% RSLogix 500 project alarm_and_notifcations.RSS, saved by version 9.00.00.04 %
PROJECT "UNTITLED"    % processor: Bul.1763 MicroLogix 1100 Series A %

PROGRAM FILES
  LAD 2 "MAIN"  10 rungs
  LAD 3 "D INPUT"  9 rungs
  LAD 4 "D OUTPUT"  6 rungs
  LAD 5 "A INPUT"  3 rungs
  LAD 6 "A OUTPUT"  2 rungs
  LAD 7 "CONTROLS"  13 rungs
  LAD 8 "ALARMS"  21 rungs
  LAD 9 "DISPLAY"  2 rungs

DATA FILES
  O0 OUTPUT  6 elements
  I1 INPUT  18 elements
  S2 STATUS  66 elements
  B3 BINARY  8 elements
  T4 TIMER  8 elements
  C5 COUNTER  1 elements
  R6 CONTROL  1 elements
  N7 INTEGER  12 elements
  F8 FLOAT  3 elements
  PD9 TEMP  1 elements

LADDER 2 "MAIN"
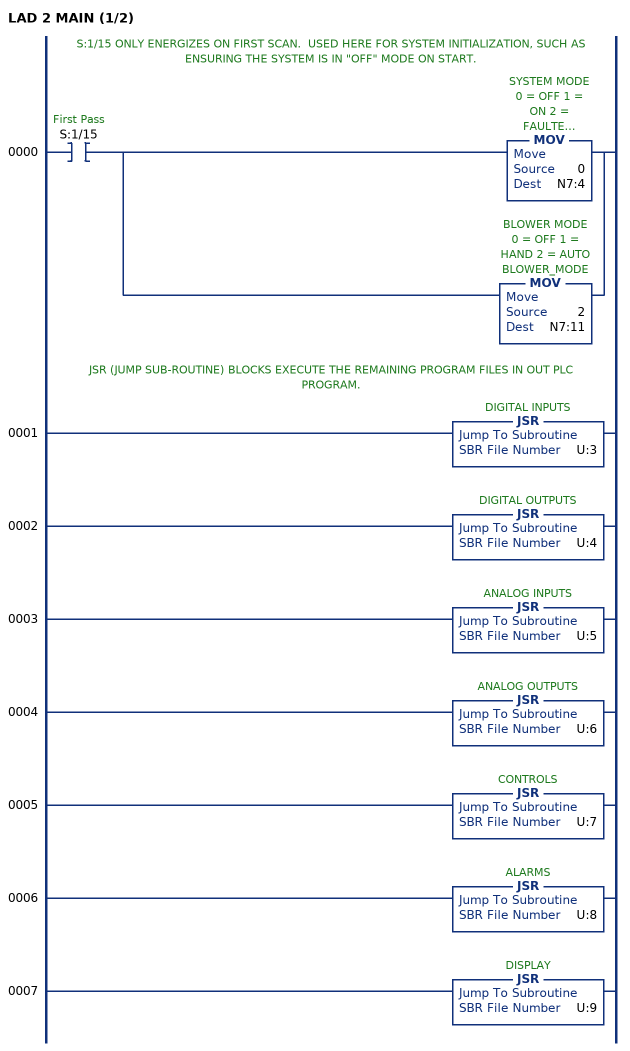
% Rung: 0 %
% S:1/15 ONLY ENERGIZES ON FIRST SCAN.  USED HERE FOR SYSTEM INITIALIZATION, SUCH AS ENSURING THE SYSTEM IS IN "OFF" MODE ON START. %
SOR XIC S:1/15 BST MOV 0 N7:4 NXB MOV 2 N7:11 BND EOR
%   S:1/15  "First Pass" %
%   N7:4  SYSTEM_MODE  "SYSTEM MODE 0 = OFF 1 = ON 2 = FAULTED" %
%   N7:11  BLOWER_MODE  "BLOWER MODE 0 = OFF 1 = HAND 2 = AUTO" %
% Rung: 1 %
% JSR (JUMP SUB-ROUTINE) BLOCKS EXECUTE THE REMAINING PROGRAM FILES IN OUT PLC PROGRAM. %
SOR JSR U:3 EOR
%   U:3  "DIGITAL INPUTS" %
% Rung: 2 %
SOR JSR U:4 EOR
%   U:4  "DIGITAL OUTPUTS" %
% Rung: 3 %
SOR JSR U:5 EOR
%   U:5  "ANALOG INPUTS" %
% Rung: 4 %
SOR JSR U:6 EOR
%   U:6  "ANALOG OUTPUTS" %
% Rung: 5 %
SOR JSR U:7 EOR
%   U:7  "CONTROLS" %
% Rung: 6 %
SOR JSR U:8 EOR
%   U:8  "ALARMS" %
% Rung: 7 %
SOR JSR U:9 EOR
%   U:9  "DISPLAY" %

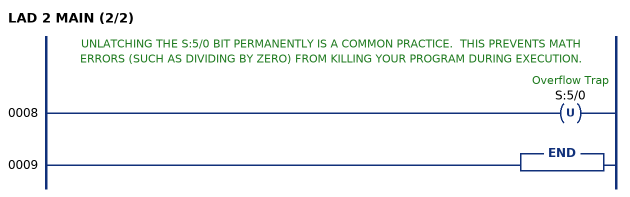
% Rung: 8 %
% UNLATCHING THE S:5/0 BIT PERMANENTLY IS A COMMON PRACTICE.  THIS PREVENTS MATH ERRORS (SUCH AS DIVIDING BY ZERO) FROM KILLING YOUR PROGRAM DURING EXECUTION. %
SOR OTU S:5/0 EOR
%   S:5/0  "Overflow Trap" %
% Rung: 9 %
SOR END EOR

LADDER 3 "D INPUT"
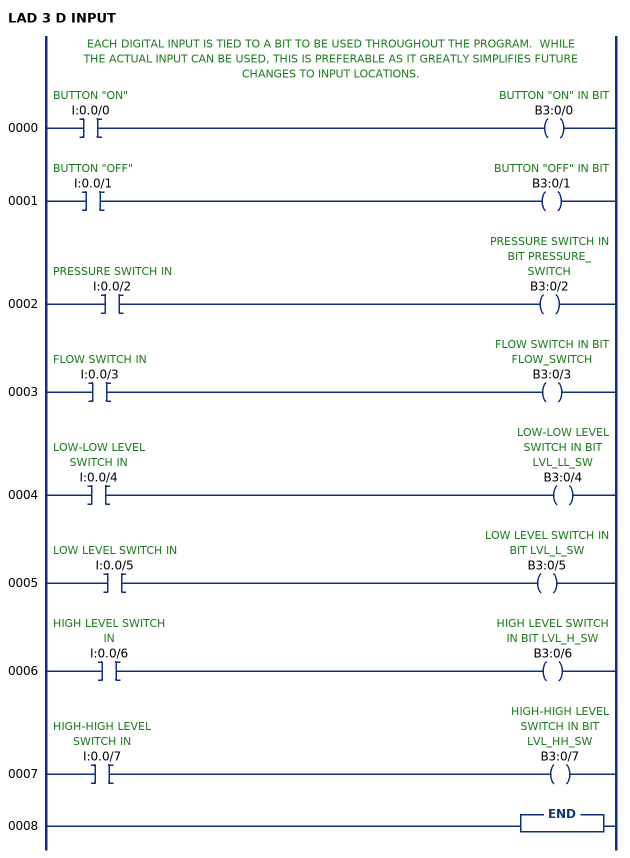
% Rung: 0 %
% EACH DIGITAL INPUT IS TIED TO A BIT TO BE USED THROUGHOUT THE PROGRAM.  WHILE THE ACTUAL INPUT CAN BE USED, THIS IS PREFERABLE AS IT GREATLY SIMPLIFIES FUTURE CHANGES TO INPUT LOCATIONS. %
SOR XIC I:0.0/0 OTE B3:0/0 EOR
%   I:0.0/0  "BUTTON "ON"" %
%   B3:0/0  "BUTTON "ON" IN BIT" %
% Rung: 1 %
SOR XIC I:0.0/1 OTE B3:0/1 EOR
%   I:0.0/1  "BUTTON "OFF"" %
%   B3:0/1  "BUTTON "OFF" IN BIT" %
% Rung: 2 %
SOR XIC I:0.0/2 OTE B3:0/2 EOR
%   I:0.0/2  "PRESSURE SWITCH IN" %
%   B3:0/2  PRESSURE_SWITCH  "PRESSURE SWITCH IN BIT" %
% Rung: 3 %
SOR XIC I:0.0/3 OTE B3:0/3 EOR
%   I:0.0/3  "FLOW SWITCH IN" %
%   B3:0/3  FLOW_SWITCH  "FLOW SWITCH IN BIT" %
% Rung: 4 %
SOR XIC I:0.0/4 OTE B3:0/4 EOR
%   I:0.0/4  "LOW-LOW LEVEL SWITCH IN" %
%   B3:0/4  LVL_LL_SW  "LOW-LOW LEVEL SWITCH IN BIT" %
% Rung: 5 %
SOR XIC I:0.0/5 OTE B3:0/5 EOR
%   I:0.0/5  "LOW LEVEL SWITCH IN" %
%   B3:0/5  LVL_L_SW  "LOW LEVEL SWITCH IN BIT" %
% Rung: 6 %
SOR XIC I:0.0/6 OTE B3:0/6 EOR
%   I:0.0/6  "HIGH LEVEL SWITCH IN" %
%   B3:0/6  LVL_H_SW  "HIGH LEVEL SWITCH IN BIT" %
% Rung: 7 %
SOR XIC I:0.0/7 OTE B3:0/7 EOR
%   I:0.0/7  "HIGH-HIGH LEVEL SWITCH IN" %
%   B3:0/7  LVL_HH_SW  "HIGH-HIGH LEVEL SWITCH IN BIT" %
% Rung: 8 %
SOR END EOR

LADDER 4 "D OUTPUT"
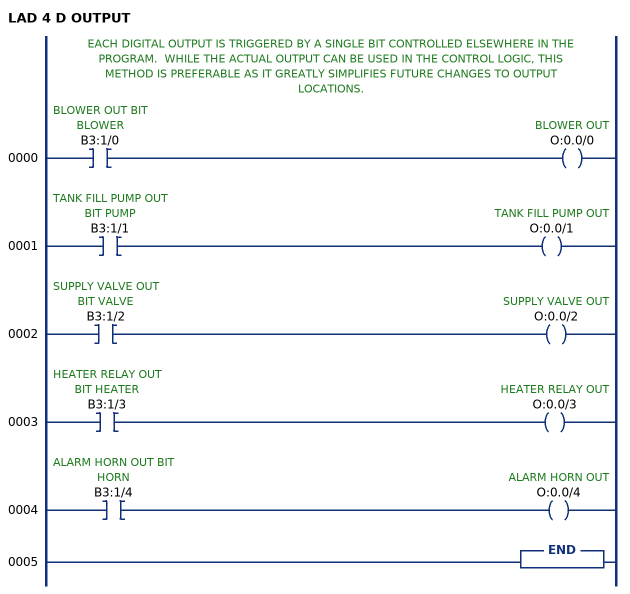
% Rung: 0 %
% EACH DIGITAL OUTPUT IS TRIGGERED BY A SINGLE BIT CONTROLLED ELSEWHERE IN THE PROGRAM.  WHILE THE ACTUAL OUTPUT CAN BE USED IN THE CONTROL LOGIC, THIS METHOD IS PREFERABLE AS IT GREATLY SIMPLIFIES FUTURE CHANGES TO OUTPUT LOCATIONS. %
SOR XIC B3:1/0 OTE O:0.0/0 EOR
%   B3:1/0  BLOWER  "BLOWER OUT BIT" %
%   O:0.0/0  "BLOWER OUT" %
% Rung: 1 %
SOR XIC B3:1/1 OTE O:0.0/1 EOR
%   B3:1/1  PUMP  "TANK FILL PUMP OUT BIT" %
%   O:0.0/1  "TANK FILL PUMP OUT" %
% Rung: 2 %
SOR XIC B3:1/2 OTE O:0.0/2 EOR
%   B3:1/2  VALVE  "SUPPLY VALVE OUT BIT" %
%   O:0.0/2  "SUPPLY VALVE OUT" %
% Rung: 3 %
SOR XIC B3:1/3 OTE O:0.0/3 EOR
%   B3:1/3  HEATER  "HEATER RELAY OUT BIT" %
%   O:0.0/3  "HEATER RELAY OUT" %
% Rung: 4 %
SOR XIC B3:1/4 OTE O:0.0/4 EOR
%   B3:1/4  HORN  "ALARM HORN OUT BIT" %
%   O:0.0/4  "ALARM HORN OUT" %
% Rung: 5 %
SOR END EOR

LADDER 5 "A INPUT"
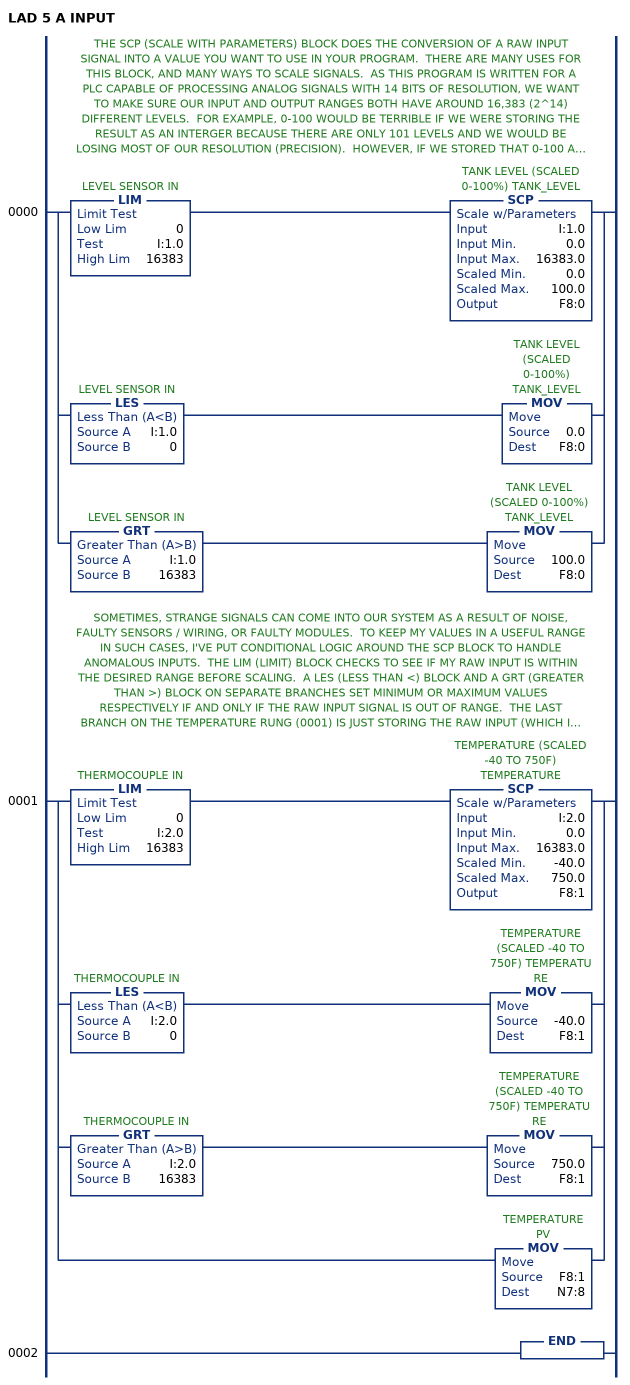
% Rung: 0 %
% THE SCP (SCALE WITH PARAMETERS) BLOCK DOES THE CONVERSION OF A RAW INPUT SIGNAL INTO A VALUE YOU WANT TO USE IN YOUR PROGRAM.  THERE ARE MANY USES FOR THIS BLOCK, AND MANY WAYS TO SCALE SIGNALS.  AS THIS PROGRAM IS WRITTEN FOR A PLC CAPABLE OF PROCESSING ANALOG SIGNALS WITH 14 BITS OF RESOLUTION, WE WANT TO MAKE SURE OUR INPUT AND OUTPUT RANGES BOTH HAVE AROUND 16,383 (2^14) DIFFERENT LEVELS.  FOR EXAMPLE, 0-100 WOULD BE TERRIBLE IF WE WERE STORING THE RESULT AS AN INTERGER BECAUSE THERE ARE ONLY 101 LEVELS AND WE WOULD BE LOSING MOST OF OUR RESOLUTION (PRECISION).  HOWEVER, IF WE STORED THAT 0-100 AS A FLOAT WITH TWO DECIMAL PLACES, IT'S BETTER BECAUSE WE THEN HAVE 10,001 LEVELS.  HOWEVER, THIS STILL ISN'T IDEAL. %
SOR BST LIM 0 I:1.0 16383 SCP I:1.0 0.0 16383.0 0.0 100.0 F8:0 NXB LES I:1.0 0 MOV 0.0 F8:0 NXB GRT I:1.0 16383 MOV 100.0 F8:0 BND EOR
%   I:1.0  "LEVEL SENSOR IN" %
%   F8:0  TANK_LEVEL  "TANK LEVEL (SCALED 0-100%)" %
% Rung: 1 %
% SOMETIMES, STRANGE SIGNALS CAN COME INTO OUR SYSTEM AS A RESULT OF NOISE, FAULTY SENSORS / WIRING, OR FAULTY MODULES.  TO KEEP MY VALUES IN A USEFUL RANGE IN SUCH CASES, I'VE PUT CONDITIONAL LOGIC AROUND THE SCP BLOCK TO HANDLE ANOMALOUS INPUTS.  THE LIM (LIMIT) BLOCK CHECKS TO SEE IF MY RAW INPUT IS WITHIN THE DESIRED RANGE BEFORE SCALING.  A LES (LESS THAN <) BLOCK AND A GRT (GREATER THAN >) BLOCK ON SEPARATE BRANCHES SET MINIMUM OR MAXIMUM VALUES RESPECTIVELY IF AND ONLY IF THE RAW INPUT SIGNAL IS OUT OF RANGE.  THE LAST BRANCH ON THE TEMPERATURE RUNG (0001) IS JUST STORING THE RAW INPUT (WHICH IS ALREADY SCALED FOR PID 0-16383) TO AN INTERGER REGISTER IN MEMORY FOR USE IN A PID CONTROL LOOP.  THIS PREVENTS ME FROM REFERRING TO THE ACTUAL INPUT WITHIN THE REST OF THE PROGRAM.  THUS, IF IN THE FUTURE WE NEED TO REMAP OUR IO, WE ONLY HAVE TO MAKE CHANGES IN THE IO PROGRAM FILES INSTEAD OF HUNTING EACH ADDRESS THROUGHOUT THE ENTIRE PROGRAM. %
SOR BST LIM 0 I:2.0 16383 SCP I:2.0 0.0 16383.0 -40.0 750.0 F8:1 NXB LES I:2.0 0 MOV -40.0 F8:1 NXB GRT I:2.0 16383 MOV 750.0 F8:1 NXB MOV F8:1 N7:8 BND EOR
%   I:2.0  "THERMOCOUPLE IN" %
%   F8:1  TEMPERATURE  "TEMPERATURE (SCALED -40 TO 750F)" %
%   N7:8  "TEMPERATURE PV" %
% Rung: 2 %
SOR END EOR

LADDER 6 "A OUTPUT"
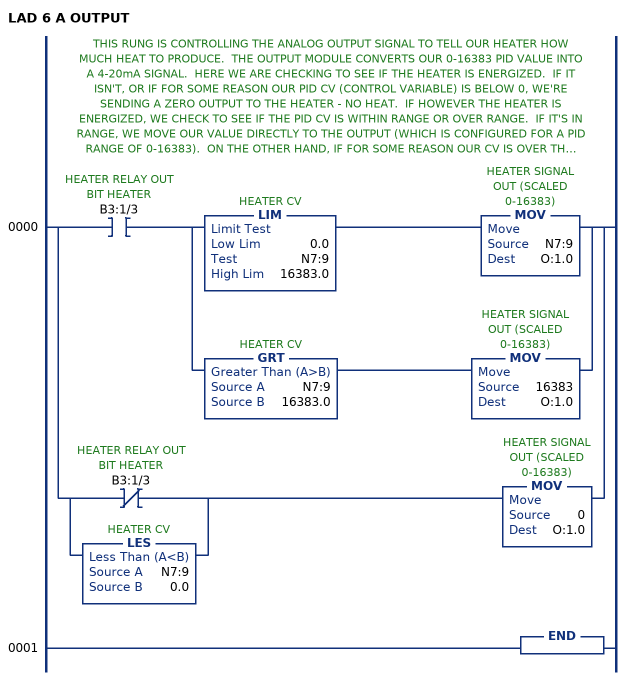
% Rung: 0 %
% THIS RUNG IS CONTROLLING THE ANALOG OUTPUT SIGNAL TO TELL OUR HEATER HOW MUCH HEAT TO PRODUCE.  THE OUTPUT MODULE CONVERTS OUR 0-16383 PID VALUE INTO A 4-20mA SIGNAL.  HERE WE ARE CHECKING TO SEE IF THE HEATER IS ENERGIZED.  IF IT ISN'T, OR IF FOR SOME REASON OUR PID CV (CONTROL VARIABLE) IS BELOW 0, WE'RE SENDING A ZERO OUTPUT TO THE HEATER - NO HEAT.  IF HOWEVER THE HEATER IS ENERGIZED, WE CHECK TO SEE IF THE PID CV IS WITHIN RANGE OR OVER RANGE.  IF IT'S IN RANGE, WE MOVE OUR VALUE DIRECTLY TO THE OUTPUT (WHICH IS CONFIGURED FOR A PID RANGE OF 0-16383).  ON THE OTHER HAND, IF FOR SOME REASON OUR CV IS OVER THE RANGE, WE'RE MOVING A MAXIMUM ACCEPTABLE VALUE TO THE OUTPUT. %
SOR BST XIC B3:1/3 BST LIM 0.0 N7:9 16383.0 MOV N7:9 O:1.0 NXB GRT N7:9 16383.0 MOV 16383 O:1.0 BND NXB BST XIO B3:1/3 NXB LES N7:9 0.0 BND MOV 0 O:1.0 BND EOR
%   B3:1/3  HEATER  "HEATER RELAY OUT BIT" %
%   N7:9  "HEATER CV" %
%   O:1.0  "HEATER SIGNAL OUT (SCALED 0-16383)" %
% Rung: 1 %
SOR END EOR

LADDER 7 "CONTROLS"
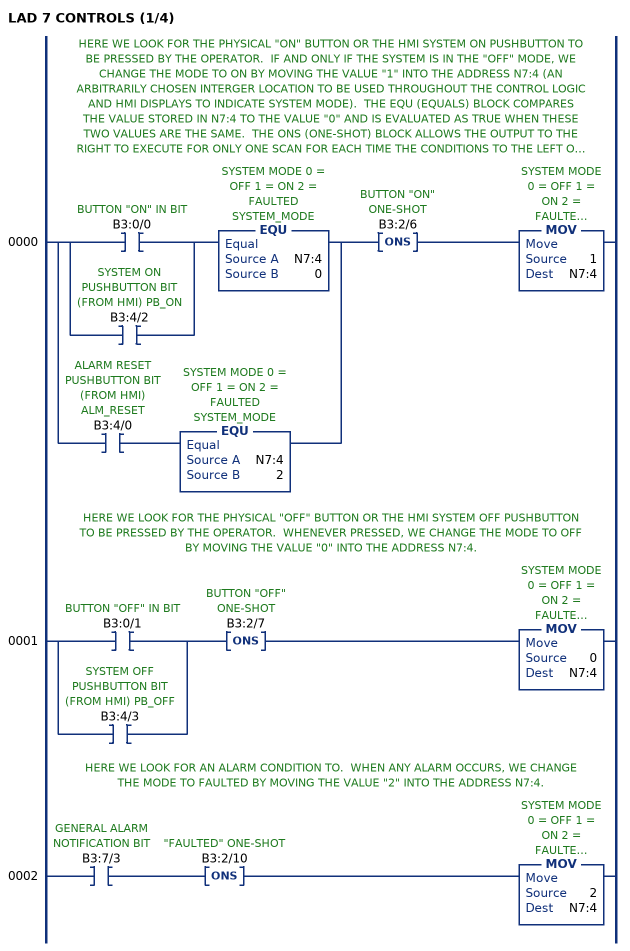
% Rung: 0 %
% HERE WE LOOK FOR THE PHYSICAL "ON" BUTTON OR THE HMI SYSTEM ON PUSHBUTTON TO BE PRESSED BY THE OPERATOR.  IF AND ONLY IF THE SYSTEM IS IN THE "OFF" MODE, WE CHANGE THE MODE TO ON BY MOVING THE VALUE "1" INTO THE ADDRESS N7:4 (AN ARBITRARILY CHOSEN INTERGER LOCATION TO BE USED THROUGHOUT THE CONTROL LOGIC AND HMI DISPLAYS TO INDICATE SYSTEM MODE).  THE EQU (EQUALS) BLOCK COMPARES THE VALUE STORED IN N7:4 TO THE VALUE "0" AND IS EVALUATED AS TRUE WHEN THESE TWO VALUES ARE THE SAME.  THE ONS (ONE-SHOT) BLOCK ALLOWS THE OUTPUT TO THE RIGHT TO EXECUTE FOR ONLY ONE SCAN FOR EACH TIME THE CONDITIONS TO THE LEFT OF THE BLOCK ARE ALL TRUE. %
SOR BST BST XIC B3:0/0 NXB XIC B3:4/2 BND EQU N7:4 0 NXB XIC B3:4/0 EQU N7:4 2 BND ONS B3:2/6 MOV 1 N7:4 EOR
%   B3:0/0  "BUTTON "ON" IN BIT" %
%   B3:4/2  PB_ON  "SYSTEM ON PUSHBUTTON BIT (FROM HMI)" %
%   N7:4  SYSTEM_MODE  "SYSTEM MODE 0 = OFF 1 = ON 2 = FAULTED" %
%   B3:4/0  ALM_RESET  "ALARM RESET PUSHBUTTON BIT (FROM HMI)" %
%   B3:2/6  "BUTTON "ON" ONE-SHOT" %
% Rung: 1 %
% HERE WE LOOK FOR THE PHYSICAL "OFF" BUTTON OR THE HMI SYSTEM OFF PUSHBUTTON TO BE PRESSED BY THE OPERATOR.  WHENEVER PRESSED, WE CHANGE THE MODE TO OFF BY MOVING THE VALUE "0" INTO THE ADDRESS N7:4. %
SOR BST XIC B3:0/1 NXB XIC B3:4/3 BND ONS B3:2/7 MOV 0 N7:4 EOR
%   B3:0/1  "BUTTON "OFF" IN BIT" %
%   B3:4/3  PB_OFF  "SYSTEM OFF PUSHBUTTON BIT (FROM HMI)" %
%   B3:2/7  "BUTTON "OFF" ONE-SHOT" %
%   N7:4  SYSTEM_MODE  "SYSTEM MODE 0 = OFF 1 = ON 2 = FAULTED" %
% Rung: 2 %
% HERE WE LOOK FOR AN ALARM CONDITION TO.  WHEN ANY ALARM OCCURS, WE CHANGE THE MODE TO FAULTED BY MOVING THE VALUE "2" INTO THE ADDRESS N7:4. %
SOR XIC B3:7/3 ONS B3:2/10 MOV 2 N7:4 EOR
%   B3:7/3  "GENERAL ALARM NOTIFICATION BIT" %
%   B3:2/10  ""FAULTED" ONE-SHOT" %
%   N7:4  SYSTEM_MODE  "SYSTEM MODE 0 = OFF 1 = ON 2 = FAULTED" %

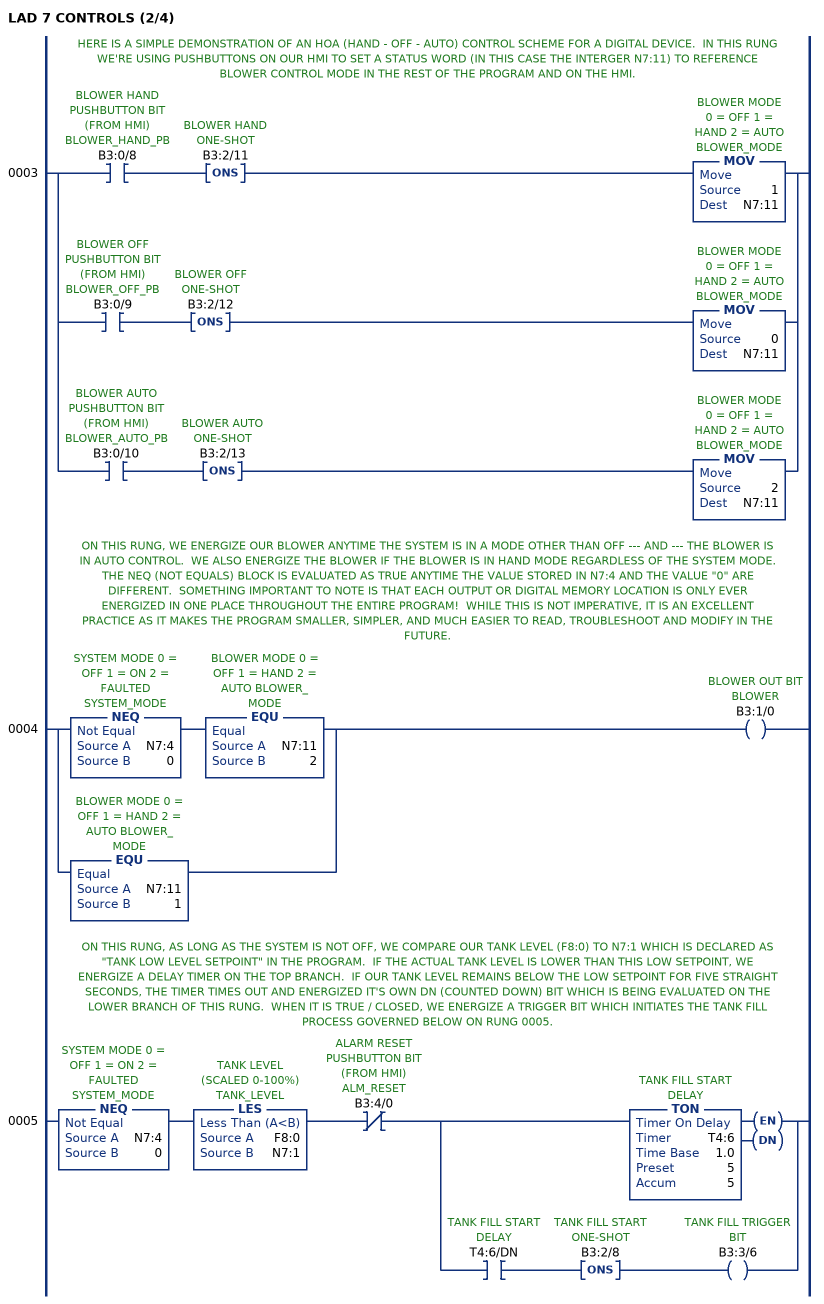
% Rung: 3 %
% HERE IS A SIMPLE DEMONSTRATION OF AN HOA (HAND - OFF - AUTO) CONTROL SCHEME FOR A DIGITAL DEVICE.  IN THIS RUNG WE'RE USING PUSHBUTTONS ON OUR HMI TO SET A STATUS WORD (IN THIS CASE THE INTERGER N7:11) TO REFERENCE BLOWER CONTROL MODE IN THE REST OF THE PROGRAM AND ON THE HMI. %
SOR BST XIC B3:0/8 ONS B3:2/11 MOV 1 N7:11 NXB XIC B3:0/9 ONS B3:2/12 MOV 0 N7:11 NXB XIC B3:0/10 ONS B3:2/13 MOV 2 N7:11 BND EOR
%   B3:0/8  BLOWER_HAND_PB  "BLOWER HAND PUSHBUTTON BIT (FROM HMI)" %
%   B3:2/11  "BLOWER HAND ONE-SHOT" %
%   N7:11  BLOWER_MODE  "BLOWER MODE 0 = OFF 1 = HAND 2 = AUTO" %
%   B3:0/9  BLOWER_OFF_PB  "BLOWER OFF PUSHBUTTON BIT (FROM HMI)" %
%   B3:2/12  "BLOWER OFF ONE-SHOT" %
%   B3:0/10  BLOWER_AUTO_PB  "BLOWER AUTO PUSHBUTTON BIT (FROM HMI)" %
%   B3:2/13  "BLOWER AUTO ONE-SHOT" %
% Rung: 4 %
% ON THIS RUNG, WE ENERGIZE OUR BLOWER ANYTIME THE SYSTEM IS IN A MODE OTHER THAN OFF --- AND --- THE BLOWER IS IN AUTO CONTROL.  WE ALSO ENERGIZE THE BLOWER IF THE BLOWER IS IN HAND MODE REGARDLESS OF THE SYSTEM MODE.  THE NEQ (NOT EQUALS) BLOCK IS EVALUATED AS TRUE ANYTIME THE VALUE STORED IN N7:4 AND THE VALUE "0" ARE DIFFERENT.  SOMETHING IMPORTANT TO NOTE IS THAT EACH OUTPUT OR DIGITAL MEMORY LOCATION IS ONLY EVER ENERGIZED IN ONE PLACE THROUGHOUT THE ENTIRE PROGRAM!  WHILE THIS IS NOT IMPERATIVE, IT IS AN EXCELLENT PRACTICE AS IT MAKES THE PROGRAM SMALLER, SIMPLER, AND MUCH EASIER TO READ, TROUBLESHOOT AND MODIFY IN THE FUTURE. %
SOR BST NEQ N7:4 0 EQU N7:11 2 NXB EQU N7:11 1 BND OTE B3:1/0 EOR
%   N7:4  SYSTEM_MODE  "SYSTEM MODE 0 = OFF 1 = ON 2 = FAULTED" %
%   N7:11  BLOWER_MODE  "BLOWER MODE 0 = OFF 1 = HAND 2 = AUTO" %
%   B3:1/0  BLOWER  "BLOWER OUT BIT" %
% Rung: 5 %
% ON THIS RUNG, AS LONG AS THE SYSTEM IS NOT OFF, WE COMPARE OUR TANK LEVEL (F8:0) TO N7:1 WHICH IS DECLARED AS "TANK LOW LEVEL SETPOINT" IN THE PROGRAM.  IF THE ACTUAL TANK LEVEL IS LOWER THAN THIS LOW SETPOINT, WE ENERGIZE A DELAY TIMER ON THE TOP BRANCH.  IF OUR TANK LEVEL REMAINS BELOW THE LOW SETPOINT FOR FIVE STRAIGHT SECONDS, THE TIMER TIMES OUT AND ENERGIZED IT'S OWN DN (COUNTED DOWN) BIT WHICH IS BEING EVALUATED ON THE LOWER BRANCH OF THIS RUNG.  WHEN IT IS TRUE / CLOSED, WE ENERGIZE A TRIGGER BIT WHICH INITIATES THE TANK FILL PROCESS GOVERNED BELOW ON RUNG 0005. %
SOR NEQ N7:4 0 LES F8:0 N7:1 XIO B3:4/0 BST TON T4:6 1.0 5 5 NXB XIC T4:6/DN ONS B3:2/8 OTE B3:3/6 BND EOR
%   N7:4  SYSTEM_MODE  "SYSTEM MODE 0 = OFF 1 = ON 2 = FAULTED" %
%   F8:0  TANK_LEVEL  "TANK LEVEL (SCALED 0-100%)" %
%   N7:1  TANK_SP_L  "TANK LOW LEVEL SETPOINT" %
%   B3:4/0  ALM_RESET  "ALARM RESET PUSHBUTTON BIT (FROM HMI)" %
%   T4:6  "TANK FILL START DELAY" %
%   B3:2/8  "TANK FILL START ONE-SHOT" %
%   B3:3/6  "TANK FILL TRIGGER BIT" %

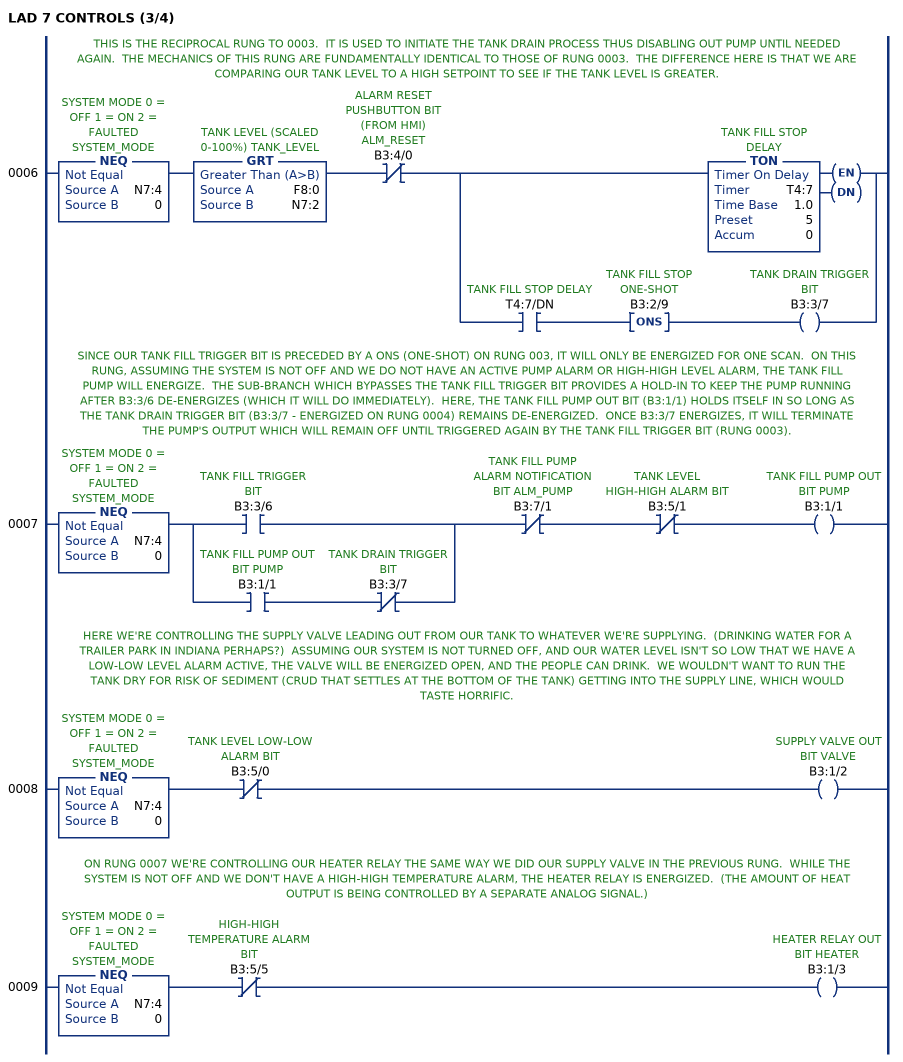
% Rung: 6 %
% THIS IS THE RECIPROCAL RUNG TO 0003.  IT IS USED TO INITIATE THE TANK DRAIN PROCESS THUS DISABLING OUT PUMP UNTIL NEEDED AGAIN.  THE MECHANICS OF THIS RUNG ARE FUNDAMENTALLY IDENTICAL TO THOSE OF RUNG 0003.  THE DIFFERENCE HERE IS THAT WE ARE COMPARING OUR TANK LEVEL TO A HIGH SETPOINT TO SEE IF THE TANK LEVEL IS GREATER. %
SOR NEQ N7:4 0 GRT F8:0 N7:2 XIO B3:4/0 BST TON T4:7 1.0 5 0 NXB XIC T4:7/DN ONS B3:2/9 OTE B3:3/7 BND EOR
%   N7:4  SYSTEM_MODE  "SYSTEM MODE 0 = OFF 1 = ON 2 = FAULTED" %
%   F8:0  TANK_LEVEL  "TANK LEVEL (SCALED 0-100%)" %
%   N7:2  TANK_SP_H  "TANK HIGH LEVEL SETPOINT" %
%   B3:4/0  ALM_RESET  "ALARM RESET PUSHBUTTON BIT (FROM HMI)" %
%   T4:7  "TANK FILL STOP DELAY" %
%   B3:2/9  "TANK FILL STOP ONE-SHOT" %
%   B3:3/7  "TANK DRAIN TRIGGER BIT" %
% Rung: 7 %
% SINCE OUR TANK FILL TRIGGER BIT IS PRECEDED BY A ONS (ONE-SHOT) ON RUNG 003, IT WILL ONLY BE ENERGIZED FOR ONE SCAN.  ON THIS RUNG, ASSUMING THE SYSTEM IS NOT OFF AND WE DO NOT HAVE AN ACTIVE PUMP ALARM OR HIGH-HIGH LEVEL ALARM, THE TANK FILL PUMP WILL ENERGIZE.  THE SUB-BRANCH WHICH BYPASSES THE TANK FILL TRIGGER BIT PROVIDES A HOLD-IN TO KEEP THE PUMP RUNNING AFTER B3:3/6 DE-ENERGIZES (WHICH IT WILL DO IMMEDIATELY).  HERE, THE TANK FILL PUMP OUT BIT (B3:1/1) HOLDS ITSELF IN SO LONG AS THE TANK DRAIN TRIGGER BIT (B3:3/7 - ENERGIZED ON RUNG 0004) REMAINS DE-ENERGIZED.  ONCE B3:3/7 ENERGIZES, IT WILL TERMINATE THE PUMP'S OUTPUT WHICH WILL REMAIN OFF UNTIL TRIGGERED AGAIN BY THE TANK FILL TRIGGER BIT (RUNG 0003). %
SOR NEQ N7:4 0 BST XIC B3:3/6 NXB XIC B3:1/1 XIO B3:3/7 BND XIO B3:7/1 XIO B3:5/1 OTE B3:1/1 EOR
%   N7:4  SYSTEM_MODE  "SYSTEM MODE 0 = OFF 1 = ON 2 = FAULTED" %
%   B3:3/6  "TANK FILL TRIGGER BIT" %
%   B3:1/1  PUMP  "TANK FILL PUMP OUT BIT" %
%   B3:3/7  "TANK DRAIN TRIGGER BIT" %
%   B3:7/1  ALM_PUMP  "TANK FILL PUMP ALARM NOTIFICATION BIT" %
%   B3:5/1  "TANK LEVEL HIGH-HIGH ALARM BIT" %
% Rung: 8 %
% HERE WE'RE CONTROLLING THE SUPPLY VALVE LEADING OUT FROM OUR TANK TO WHATEVER WE'RE SUPPLYING.  (DRINKING WATER FOR A TRAILER PARK IN INDIANA PERHAPS?)  ASSUMING OUR SYSTEM IS NOT TURNED OFF, AND OUR WATER LEVEL ISN'T SO LOW THAT WE HAVE A LOW-LOW LEVEL ALARM ACTIVE, THE VALVE WILL BE ENERGIZED OPEN, AND THE PEOPLE CAN DRINK.  WE WOULDN'T WANT TO RUN THE TANK DRY FOR RISK OF SEDIMENT (CRUD THAT SETTLES AT THE BOTTOM OF THE TANK) GETTING INTO THE SUPPLY LINE, WHICH WOULD TASTE HORRIFIC. %
SOR NEQ N7:4 0 XIO B3:5/0 OTE B3:1/2 EOR
%   N7:4  SYSTEM_MODE  "SYSTEM MODE 0 = OFF 1 = ON 2 = FAULTED" %
%   B3:5/0  "TANK LEVEL LOW-LOW ALARM BIT" %
%   B3:1/2  VALVE  "SUPPLY VALVE OUT BIT" %
% Rung: 9 %
% ON RUNG 0007 WE'RE CONTROLLING OUR HEATER RELAY THE SAME WAY WE DID OUR SUPPLY VALVE IN THE PREVIOUS RUNG.  WHILE THE SYSTEM IS NOT OFF AND WE DON'T HAVE A HIGH-HIGH TEMPERATURE ALARM, THE HEATER RELAY IS ENERGIZED.  (THE AMOUNT OF HEAT OUTPUT IS BEING CONTROLLED BY A SEPARATE ANALOG SIGNAL.) %
SOR NEQ N7:4 0 XIO B3:5/5 OTE B3:1/3 EOR
%   N7:4  SYSTEM_MODE  "SYSTEM MODE 0 = OFF 1 = ON 2 = FAULTED" %
%   B3:5/5  "HIGH-HIGH TEMPERATURE ALARM BIT" %
%   B3:1/3  HEATER  "HEATER RELAY OUT BIT" %

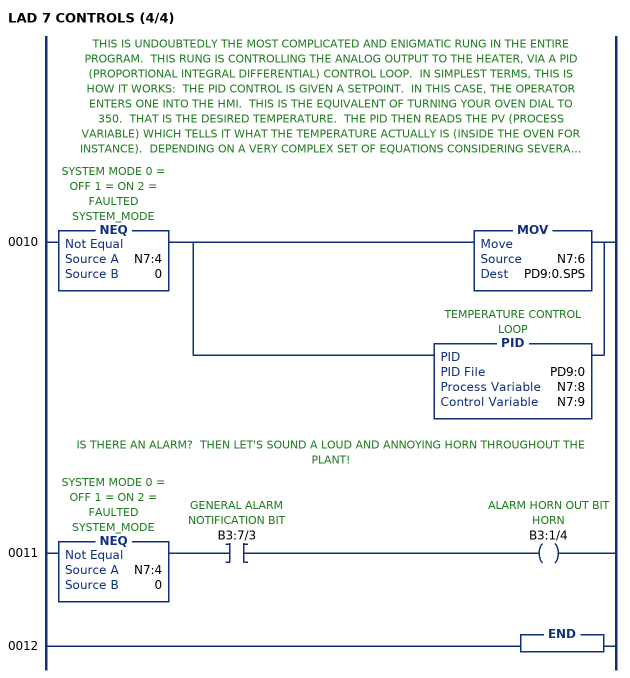
% Rung: 10 %
% THIS IS UNDOUBTEDLY THE MOST COMPLICATED AND ENIGMATIC RUNG IN THE ENTIRE PROGRAM.  THIS RUNG IS CONTROLLING THE ANALOG OUTPUT TO THE HEATER, VIA A PID (PROPORTIONAL INTEGRAL DIFFERENTIAL) CONTROL LOOP.  IN SIMPLEST TERMS, THIS IS HOW IT WORKS:  THE PID CONTROL IS GIVEN A SETPOINT.  IN THIS CASE, THE OPERATOR ENTERS ONE INTO THE HMI.  THIS IS THE EQUIVALENT OF TURNING YOUR OVEN DIAL TO 350.  THAT IS THE DESIRED TEMPERATURE.  THE PID THEN READS THE PV (PROCESS VARIABLE) WHICH TELLS IT WHAT THE TEMPERATURE ACTUALLY IS (INSIDE THE OVEN FOR INSTANCE).  DEPENDING ON A VERY COMPLEX SET OF EQUATIONS CONSIDERING SEVERAL PROGRAMMER-CONFIGURABLE VARIABLES TOO COMPLEX TO GET INTO IN THIS TUTORIAL, IT ADJUSTS THE CV (CONTROL VARIABLE) UP OR DOWN TO TRY TO MAINTAIN THE TEMPERATURE AT THE SETPOINT.  THE CV IS WHAT WE USE IN THE ANALOG OUTPUT PROGRAM FILE TO ESTABLISH A SIGNAL TO SEND TO THE HEATER.  THE MOV (MOVE) BLOCK HERE IS JUST STORING THE OPERATOR'S SETPOINT INTO THE PID SO IT CAN BE EVALUATED THERE.  THERE ARE BOOKS, PROGRAMS AND ENTIRE COURSES ON HOW TO SETUP AND 'TUNE' PID'S.  FOR SMALLER APPLICATIONS OR APPLICATIONS BEING USED BY LESS-THAN-FLUENT OPERATORS, MANY PROGRAMMERS RIGHTLY SHY AWAY FROM USING PID'S TO CONTROL PROCESS IN ALL BUT CRITICAL PROCESSES. %
SOR NEQ N7:4 0 BST MOV N7:6 PD9:0.SPS NXB PID PD9:0 N7:8 N7:9 BND EOR
%   N7:4  SYSTEM_MODE  "SYSTEM MODE 0 = OFF 1 = ON 2 = FAULTED" %
%   N7:6  TEMP_SP  "TEMPERATURE SETPOINT" %
%   PD9:0  "TEMPERATURE CONTROL LOOP" %
%   N7:8  "TEMPERATURE PV" %
%   N7:9  "HEATER CV" %
% Rung: 11 %
% IS THERE AN ALARM?  THEN LET'S SOUND A LOUD AND ANNOYING HORN THROUGHOUT THE PLANT! %
SOR NEQ N7:4 0 XIC B3:7/3 OTE B3:1/4 EOR
%   N7:4  SYSTEM_MODE  "SYSTEM MODE 0 = OFF 1 = ON 2 = FAULTED" %
%   B3:7/3  "GENERAL ALARM NOTIFICATION BIT" %
%   B3:1/4  HORN  "ALARM HORN OUT BIT" %
% Rung: 12 %
SOR END EOR

LADDER 8 "ALARMS"
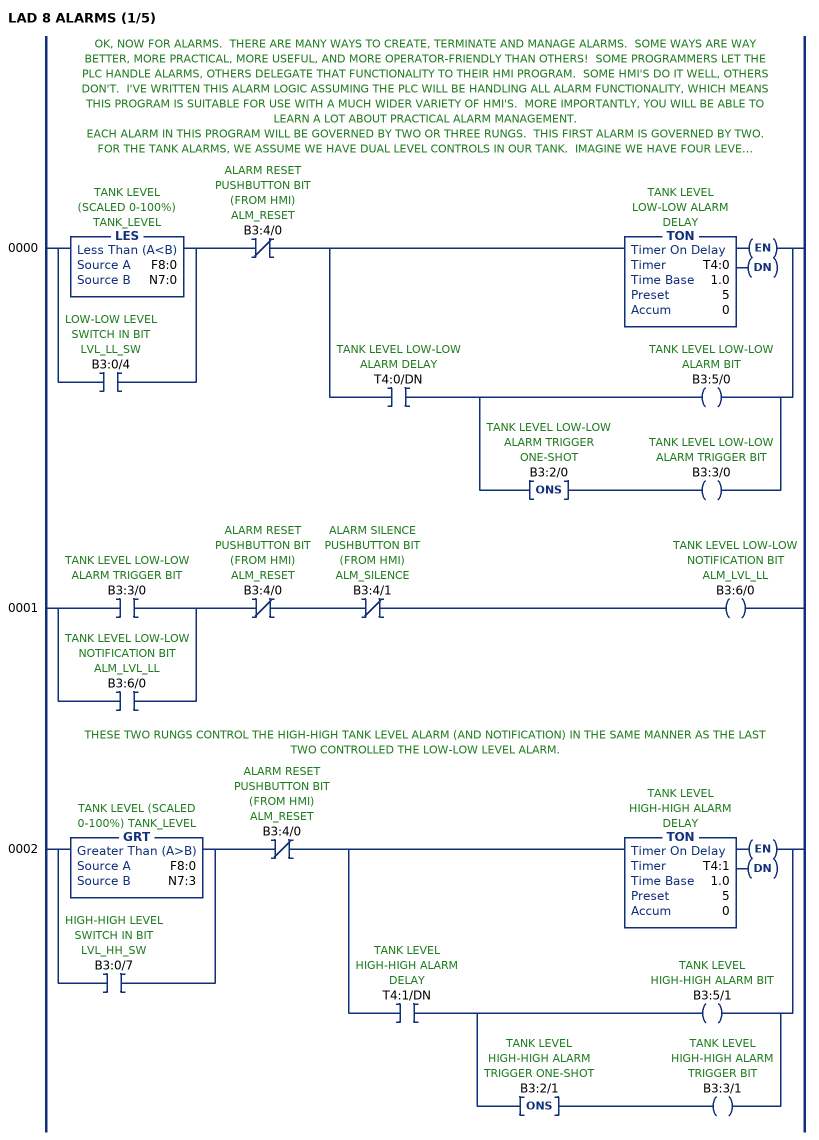
% Rung: 0 %
% OK, NOW FOR ALARMS.  THERE ARE MANY WAYS TO CREATE, TERMINATE AND MANAGE ALARMS.  SOME WAYS ARE WAY BETTER, MORE PRACTICAL, MORE USEFUL, AND MORE OPERATOR-FRIENDLY THAN OTHERS!  SOME PROGRAMMERS LET THE PLC HANDLE ALARMS, OTHERS DELEGATE THAT FUNCTIONALITY TO THEIR HMI PROGRAM.  SOME HMI'S DO IT WELL, OTHERS DON'T.  I'VE WRITTEN THIS ALARM LOGIC ASSUMING THE PLC WILL BE HANDLING ALL ALARM FUNCTIONALITY, WHICH MEANS THIS PROGRAM IS SUITABLE FOR USE WITH A MUCH WIDER VARIETY OF HMI'S.  MORE IMPORTANTLY, YOU WILL BE ABLE TO LEARN A LOT ABOUT PRACTICAL ALARM MANAGEMENT.
% 
% EACH ALARM IN THIS PROGRAM WILL BE GOVERNED BY TWO OR THREE RUNGS.  THIS FIRST ALARM IS GOVERNED BY TWO.  FOR THE TANK ALARMS, WE ASSUME WE HAVE DUAL LEVEL CONTROLS IN OUR TANK.  IMAGINE WE HAVE FOUR LEVEL SWITCHES (FLOAT SWITCHES), ONE AT THE LOW-LOW LEVEL, ONE AT THE LOW LEVEL, ONE AT THE HIGH LEVEL AND ANOTHER AT THE HIGH-HIGH LEVEL.  WE ALSO HAVE AN ANALOG SENSOR (RADAR OR HYDROSTATIC PRESSURE FOR INSTANCE).  ON THE LEFT OF OUR RUNG, WE ARE EXAMINING BOTH CONTROLS, EITHER OF WHICH CAN TELL US WE HAVE A LOW-LOW LEVEL.  IF OUR ANALOG-MEASURED TANK LEVEL (F8:0) IS LOWER THAN OUR LOW-LOW LEVEL SETPOINT (STORED IN N7:0), --- OR --- IF OUR LOW-LOW LEVEL SWITCH IS CLOSED, THEN WE ENERGIZE OUR DELAY TIMER.  ONCE THE FIVE SECONDS ON THE TIMER EXPIRE, WE'LL TRIGGER OUR LOW-LOW ALARM BIT  --- AND --- A SEPARATE LOW-LOW NOTIFICATION BIT (IN THE RUNG BELOW - 0001) USING THE FAMILIAR ONE-SHOT AND TRIGGER BIT (JUST LIKE WE USED IN CONTROLS 0004 AND 0005).
% 
% IN THIS ALARM, ONCE THE LOW-LOW LEVEL CONDITION DISAPPEARS, THE ALARM DOES AS WELL - AUTOMATICALLY, --- BUT --- THE NOTIFICATION REMAINS!!!  WHY?  IF A LEVEL ALARM OCCURS AT 3 O'CLOCK IN THE MORNING AND THEN FIXES ITSELF, DO WE WANT TO SHUT THE SYSTEM DOWN UNTIL SOMEBODY SHOWS UP AT TEN?  MEANWHILE, A LOT OF PEOPLE HAVE NO WATER.  OF COURSE NOT.  SO WE'LL LET THE ALARM CLEAR ITSELF, --- BUT --- WE WANT THE NOTIFICATION TO STILL BE THERE WHEN THE OPERATOR SHOWS UP FOR WORK.  THAT WAY, HE CAN SEE THAT SOMETHING NEEDS HIS ATTENTION.  THE NOTIFICATION BIT REMAINS ENERGIZED UNTIL HE PRESSES THE ALARM RESET --- OR --- THE ALARM SILENCE BUTTON ON THE HMI.  THESE ARE DIFFERENT.  ONE (ALARM SILENCE) MAKES THE HORNS SHUT OFF AND THE MESSAGES ON THE HMI DISAPPEAR.  THE OTHER (ALARM RESET) CAN ACTUALLY RESET ALARMS THAT ARE LOCKED IN.  THE ALARM RESET WILL ALSO RESET THE ALARM TIMERS AND MAKE THE ALARMS DISAPPEAR --- HOWEVER --- IF THE CONDITION THAT PRECIPITATED THE ALARM REMAINS, THE ALARM AND NOTIFICATION WILL REAPPEAR ONCE THE DELAY TIMER COUNTS DOWN ANEW.
% 
% WE WON'T BE LOCKING OUR LEVEL ALARMS IN, BUT YOU CAN BET WE'LL BE LOCKING IN OUR PUMP AND TEMPERATURE ALARMS!  THOSE CAN BECOME EXPENSIVE / DANGEROUS IF LEFT UNATTENDED (AS COULD LEVEL ALARMS IF THE TANK WAS STORING BATTERY ACID OR ANTHRAX SPORES OR SOMETHING...) %
SOR BST LES F8:0 N7:0 NXB XIC B3:0/4 BND XIO B3:4/0 BST TON T4:0 1.0 5 0 NXB XIC T4:0/DN BST OTE B3:5/0 NXB ONS B3:2/0 OTE B3:3/0 BND BND EOR
%   F8:0  TANK_LEVEL  "TANK LEVEL (SCALED 0-100%)" %
%   N7:0  TANK_SP_LL  "TANK LOW-LOW LEVEL SETPOINT" %
%   B3:0/4  LVL_LL_SW  "LOW-LOW LEVEL SWITCH IN BIT" %
%   B3:4/0  ALM_RESET  "ALARM RESET PUSHBUTTON BIT (FROM HMI)" %
%   T4:0  "TANK LEVEL LOW-LOW ALARM DELAY" %
%   B3:5/0  "TANK LEVEL LOW-LOW ALARM BIT" %
%   B3:2/0  "TANK LEVEL LOW-LOW ALARM TRIGGER ONE-SHOT" %
%   B3:3/0  "TANK LEVEL LOW-LOW ALARM TRIGGER BIT" %
% Rung: 1 %
SOR BST XIC B3:3/0 NXB XIC B3:6/0 BND XIO B3:4/0 XIO B3:4/1 OTE B3:6/0 EOR
%   B3:3/0  "TANK LEVEL LOW-LOW ALARM TRIGGER BIT" %
%   B3:6/0  ALM_LVL_LL  "TANK LEVEL LOW-LOW NOTIFICATION BIT" %
%   B3:4/0  ALM_RESET  "ALARM RESET PUSHBUTTON BIT (FROM HMI)" %
%   B3:4/1  ALM_SILENCE  "ALARM SILENCE PUSHBUTTON BIT (FROM HMI)" %
% Rung: 2 %
% THESE TWO RUNGS CONTROL THE HIGH-HIGH TANK LEVEL ALARM (AND NOTIFICATION) IN THE SAME MANNER AS THE LAST TWO CONTROLLED THE LOW-LOW LEVEL ALARM. %
SOR BST GRT F8:0 N7:3 NXB XIC B3:0/7 BND XIO B3:4/0 BST TON T4:1 1.0 5 0 NXB XIC T4:1/DN BST OTE B3:5/1 NXB ONS B3:2/1 OTE B3:3/1 BND BND EOR
%   F8:0  TANK_LEVEL  "TANK LEVEL (SCALED 0-100%)" %
%   N7:3  TANK_SP_HH  "TANK HIGH-HIGH LEVEL SETPOINT" %
%   B3:0/7  LVL_HH_SW  "HIGH-HIGH LEVEL SWITCH IN BIT" %
%   B3:4/0  ALM_RESET  "ALARM RESET PUSHBUTTON BIT (FROM HMI)" %
%   T4:1  "TANK LEVEL HIGH-HIGH ALARM DELAY" %
%   B3:5/1  "TANK LEVEL HIGH-HIGH ALARM BIT" %
%   B3:2/1  "TANK LEVEL HIGH-HIGH ALARM TRIGGER ONE-SHOT" %
%   B3:3/1  "TANK LEVEL HIGH-HIGH ALARM TRIGGER BIT" %

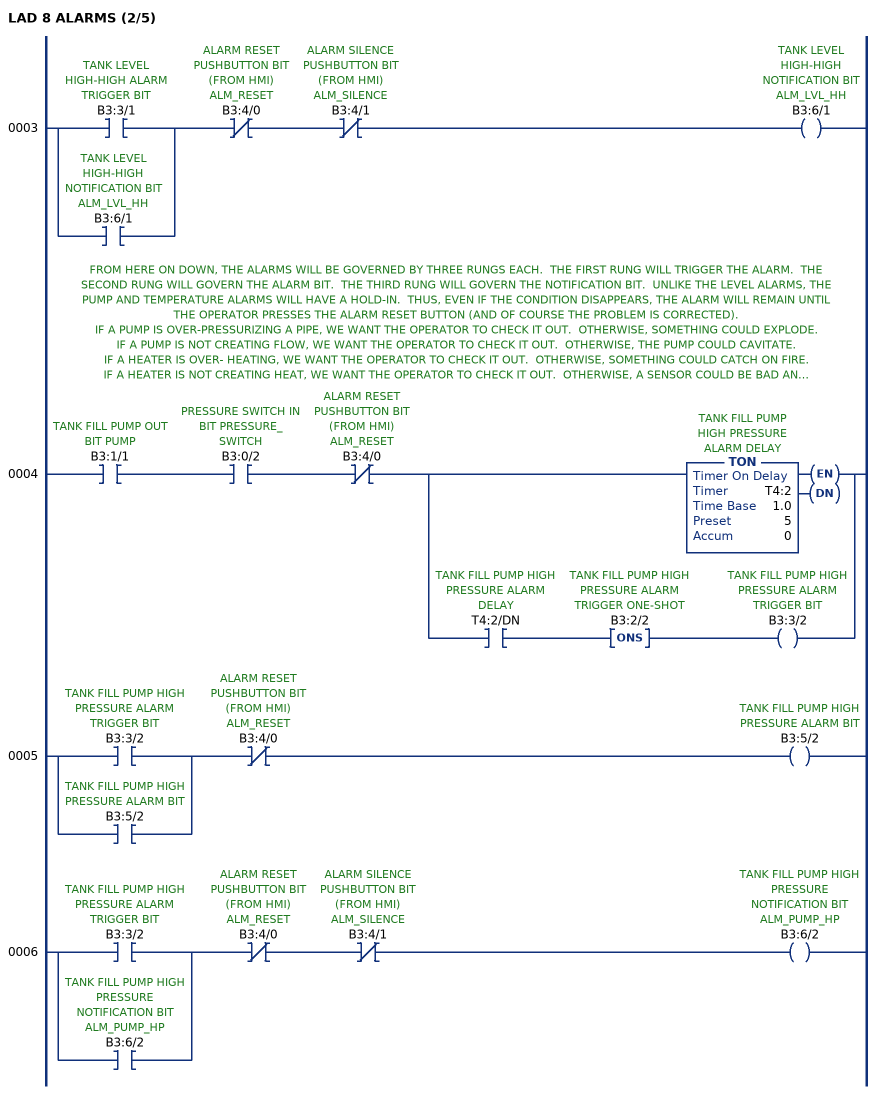
% Rung: 3 %
SOR BST XIC B3:3/1 NXB XIC B3:6/1 BND XIO B3:4/0 XIO B3:4/1 OTE B3:6/1 EOR
%   B3:3/1  "TANK LEVEL HIGH-HIGH ALARM TRIGGER BIT" %
%   B3:6/1  ALM_LVL_HH  "TANK LEVEL HIGH-HIGH NOTIFICATION BIT" %
%   B3:4/0  ALM_RESET  "ALARM RESET PUSHBUTTON BIT (FROM HMI)" %
%   B3:4/1  ALM_SILENCE  "ALARM SILENCE PUSHBUTTON BIT (FROM HMI)" %
% Rung: 4 %
% FROM HERE ON DOWN, THE ALARMS WILL BE GOVERNED BY THREE RUNGS EACH.  THE FIRST RUNG WILL TRIGGER THE ALARM.  THE SECOND RUNG WILL GOVERN THE ALARM BIT.  THE THIRD RUNG WILL GOVERN THE NOTIFICATION BIT.  UNLIKE THE LEVEL ALARMS, THE PUMP AND TEMPERATURE ALARMS WILL HAVE A HOLD-IN.  THUS, EVEN IF THE CONDITION DISAPPEARS, THE ALARM WILL REMAIN UNTIL THE OPERATOR PRESSES THE ALARM RESET BUTTON (AND OF COURSE THE PROBLEM IS CORRECTED).
% 
% IF A PUMP IS OVER-PRESSURIZING A PIPE, WE WANT THE OPERATOR TO CHECK IT OUT.  OTHERWISE, SOMETHING COULD EXPLODE.
% IF A PUMP IS NOT CREATING FLOW, WE WANT THE OPERATOR TO CHECK IT OUT.  OTHERWISE, THE PUMP COULD CAVITATE.
% IF A HEATER IS OVER- HEATING, WE WANT THE OPERATOR TO CHECK IT OUT.  OTHERWISE, SOMETHING COULD CATCH ON FIRE.
% IF A HEATER IS NOT CREATING HEAT, WE WANT THE OPERATOR TO CHECK IT OUT.  OTHERWISE, A SENSOR COULD BE BAD AND SOMETHING COULD EXPLODE. %
SOR XIC B3:1/1 XIC B3:0/2 XIO B3:4/0 BST TON T4:2 1.0 5 0 NXB XIC T4:2/DN ONS B3:2/2 OTE B3:3/2 BND EOR
%   B3:1/1  PUMP  "TANK FILL PUMP OUT BIT" %
%   B3:0/2  PRESSURE_SWITCH  "PRESSURE SWITCH IN BIT" %
%   B3:4/0  ALM_RESET  "ALARM RESET PUSHBUTTON BIT (FROM HMI)" %
%   T4:2  "TANK FILL PUMP HIGH PRESSURE ALARM DELAY" %
%   B3:2/2  "TANK FILL PUMP HIGH PRESSURE ALARM TRIGGER ONE-SHOT" %
%   B3:3/2  "TANK FILL PUMP HIGH PRESSURE ALARM TRIGGER BIT" %
% Rung: 5 %
SOR BST XIC B3:3/2 NXB XIC B3:5/2 BND XIO B3:4/0 OTE B3:5/2 EOR
%   B3:3/2  "TANK FILL PUMP HIGH PRESSURE ALARM TRIGGER BIT" %
%   B3:5/2  "TANK FILL PUMP HIGH PRESSURE ALARM BIT" %
%   B3:4/0  ALM_RESET  "ALARM RESET PUSHBUTTON BIT (FROM HMI)" %
% Rung: 6 %
SOR BST XIC B3:3/2 NXB XIC B3:6/2 BND XIO B3:4/0 XIO B3:4/1 OTE B3:6/2 EOR
%   B3:3/2  "TANK FILL PUMP HIGH PRESSURE ALARM TRIGGER BIT" %
%   B3:6/2  ALM_PUMP_HP  "TANK FILL PUMP HIGH PRESSURE NOTIFICATION BIT" %
%   B3:4/0  ALM_RESET  "ALARM RESET PUSHBUTTON BIT (FROM HMI)" %
%   B3:4/1  ALM_SILENCE  "ALARM SILENCE PUSHBUTTON BIT (FROM HMI)" %

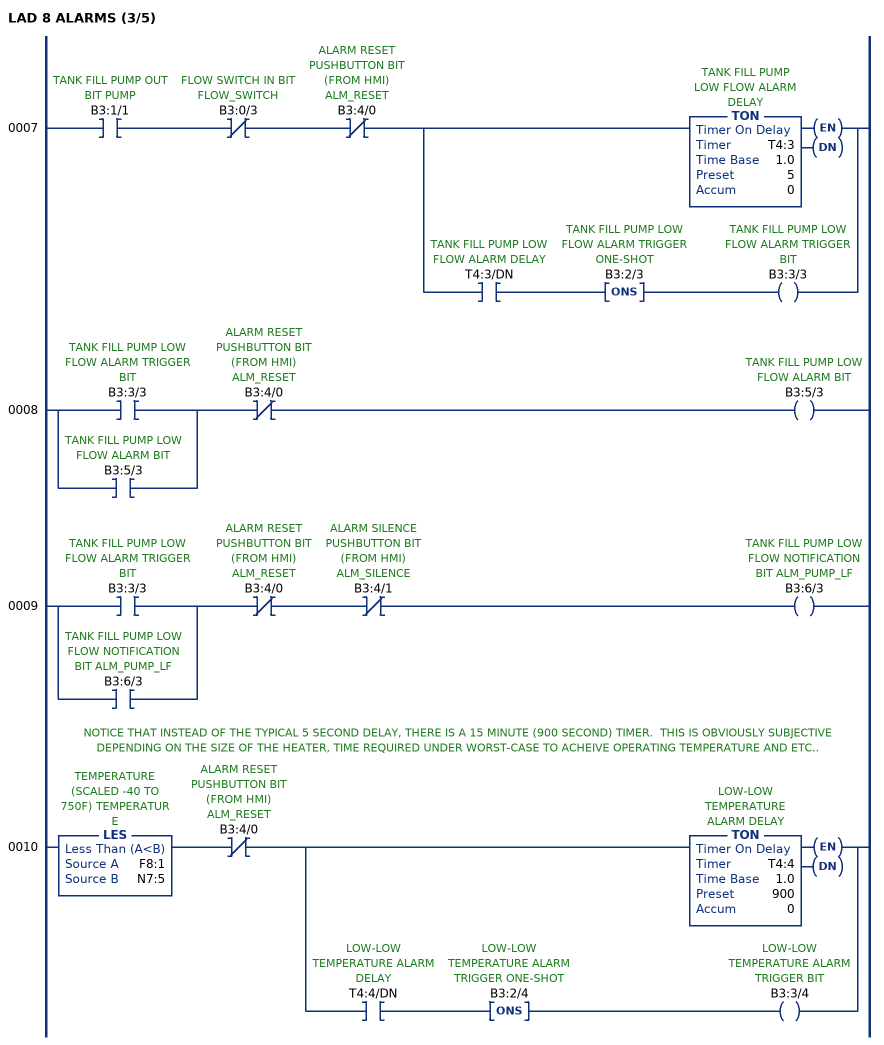
% Rung: 7 %
SOR XIC B3:1/1 XIO B3:0/3 XIO B3:4/0 BST TON T4:3 1.0 5 0 NXB XIC T4:3/DN ONS B3:2/3 OTE B3:3/3 BND EOR
%   B3:1/1  PUMP  "TANK FILL PUMP OUT BIT" %
%   B3:0/3  FLOW_SWITCH  "FLOW SWITCH IN BIT" %
%   B3:4/0  ALM_RESET  "ALARM RESET PUSHBUTTON BIT (FROM HMI)" %
%   T4:3  "TANK FILL PUMP LOW FLOW ALARM DELAY" %
%   B3:2/3  "TANK FILL PUMP LOW FLOW ALARM TRIGGER ONE-SHOT" %
%   B3:3/3  "TANK FILL PUMP LOW FLOW ALARM TRIGGER BIT" %
% Rung: 8 %
SOR BST XIC B3:3/3 NXB XIC B3:5/3 BND XIO B3:4/0 OTE B3:5/3 EOR
%   B3:3/3  "TANK FILL PUMP LOW FLOW ALARM TRIGGER BIT" %
%   B3:5/3  "TANK FILL PUMP LOW FLOW ALARM BIT" %
%   B3:4/0  ALM_RESET  "ALARM RESET PUSHBUTTON BIT (FROM HMI)" %
% Rung: 9 %
SOR BST XIC B3:3/3 NXB XIC B3:6/3 BND XIO B3:4/0 XIO B3:4/1 OTE B3:6/3 EOR
%   B3:3/3  "TANK FILL PUMP LOW FLOW ALARM TRIGGER BIT" %
%   B3:6/3  ALM_PUMP_LF  "TANK FILL PUMP LOW FLOW NOTIFICATION BIT" %
%   B3:4/0  ALM_RESET  "ALARM RESET PUSHBUTTON BIT (FROM HMI)" %
%   B3:4/1  ALM_SILENCE  "ALARM SILENCE PUSHBUTTON BIT (FROM HMI)" %
% Rung: 10 %
% NOTICE THAT INSTEAD OF THE TYPICAL 5 SECOND DELAY, THERE IS A 15 MINUTE (900 SECOND) TIMER.  THIS IS OBVIOUSLY SUBJECTIVE DEPENDING ON THE SIZE OF THE HEATER, TIME REQUIRED UNDER WORST-CASE TO ACHEIVE OPERATING TEMPERATURE AND ETC.. %
SOR LES F8:1 N7:5 XIO B3:4/0 BST TON T4:4 1.0 900 0 NXB XIC T4:4/DN ONS B3:2/4 OTE B3:3/4 BND EOR
%   F8:1  TEMPERATURE  "TEMPERATURE (SCALED -40 TO 750F)" %
%   N7:5  TEMP_SP_LL  "TEMPERATURE LOW-LOW SETPOINT" %
%   B3:4/0  ALM_RESET  "ALARM RESET PUSHBUTTON BIT (FROM HMI)" %
%   T4:4  "LOW-LOW TEMPERATURE ALARM DELAY" %
%   B3:2/4  "LOW-LOW TEMPERATURE ALARM TRIGGER ONE-SHOT" %
%   B3:3/4  "LOW-LOW TEMPERATURE ALARM TRIGGER BIT" %

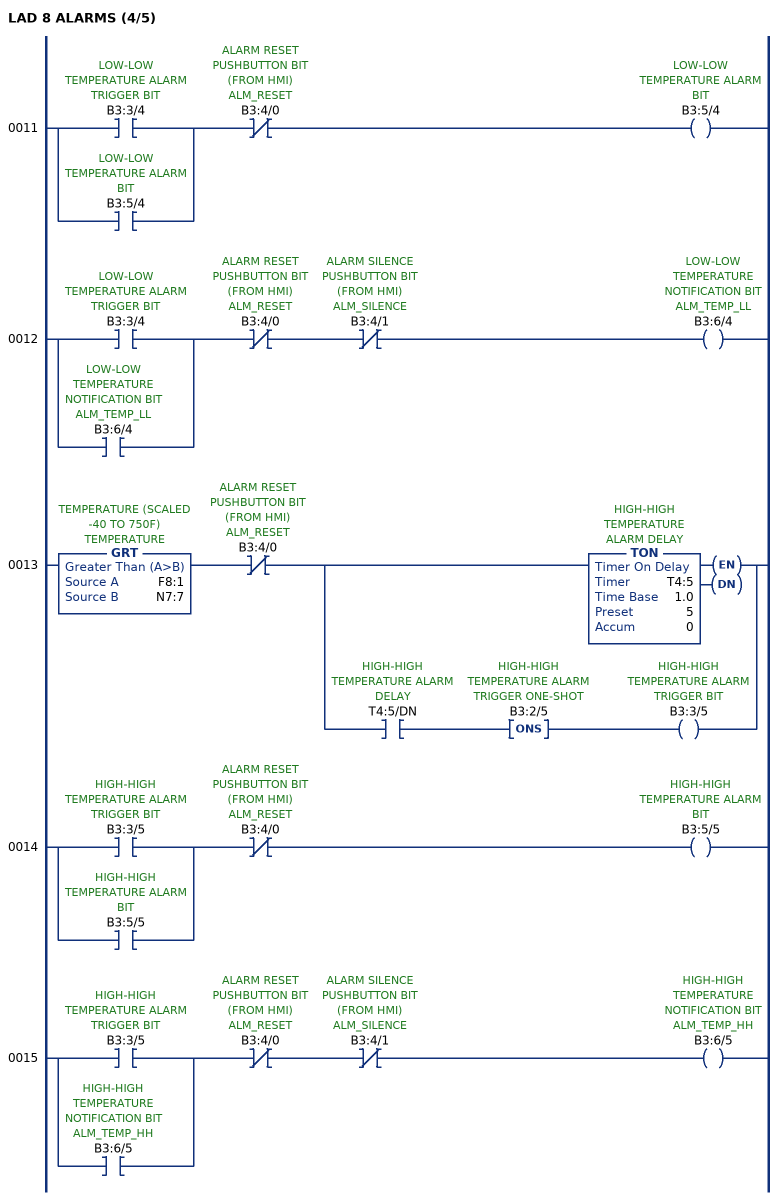
% Rung: 11 %
SOR BST XIC B3:3/4 NXB XIC B3:5/4 BND XIO B3:4/0 OTE B3:5/4 EOR
%   B3:3/4  "LOW-LOW TEMPERATURE ALARM TRIGGER BIT" %
%   B3:5/4  "LOW-LOW TEMPERATURE ALARM BIT" %
%   B3:4/0  ALM_RESET  "ALARM RESET PUSHBUTTON BIT (FROM HMI)" %
% Rung: 12 %
SOR BST XIC B3:3/4 NXB XIC B3:6/4 BND XIO B3:4/0 XIO B3:4/1 OTE B3:6/4 EOR
%   B3:3/4  "LOW-LOW TEMPERATURE ALARM TRIGGER BIT" %
%   B3:6/4  ALM_TEMP_LL  "LOW-LOW TEMPERATURE NOTIFICATION BIT" %
%   B3:4/0  ALM_RESET  "ALARM RESET PUSHBUTTON BIT (FROM HMI)" %
%   B3:4/1  ALM_SILENCE  "ALARM SILENCE PUSHBUTTON BIT (FROM HMI)" %
% Rung: 13 %
SOR GRT F8:1 N7:7 XIO B3:4/0 BST TON T4:5 1.0 5 0 NXB XIC T4:5/DN ONS B3:2/5 OTE B3:3/5 BND EOR
%   F8:1  TEMPERATURE  "TEMPERATURE (SCALED -40 TO 750F)" %
%   N7:7  TEMP_SP_HH  "TEMPERATURE HIGH- HIGH SETPOINT" %
%   B3:4/0  ALM_RESET  "ALARM RESET PUSHBUTTON BIT (FROM HMI)" %
%   T4:5  "HIGH-HIGH TEMPERATURE ALARM DELAY" %
%   B3:2/5  "HIGH-HIGH TEMPERATURE ALARM TRIGGER ONE-SHOT" %
%   B3:3/5  "HIGH-HIGH TEMPERATURE ALARM TRIGGER BIT" %
% Rung: 14 %
SOR BST XIC B3:3/5 NXB XIC B3:5/5 BND XIO B3:4/0 OTE B3:5/5 EOR
%   B3:3/5  "HIGH-HIGH TEMPERATURE ALARM TRIGGER BIT" %
%   B3:5/5  "HIGH-HIGH TEMPERATURE ALARM BIT" %
%   B3:4/0  ALM_RESET  "ALARM RESET PUSHBUTTON BIT (FROM HMI)" %
% Rung: 15 %
SOR BST XIC B3:3/5 NXB XIC B3:6/5 BND XIO B3:4/0 XIO B3:4/1 OTE B3:6/5 EOR
%   B3:3/5  "HIGH-HIGH TEMPERATURE ALARM TRIGGER BIT" %
%   B3:6/5  ALM_TEMP_HH  "HIGH-HIGH TEMPERATURE NOTIFICATION BIT" %
%   B3:4/0  ALM_RESET  "ALARM RESET PUSHBUTTON BIT (FROM HMI)" %
%   B3:4/1  ALM_SILENCE  "ALARM SILENCE PUSHBUTTON BIT (FROM HMI)" %

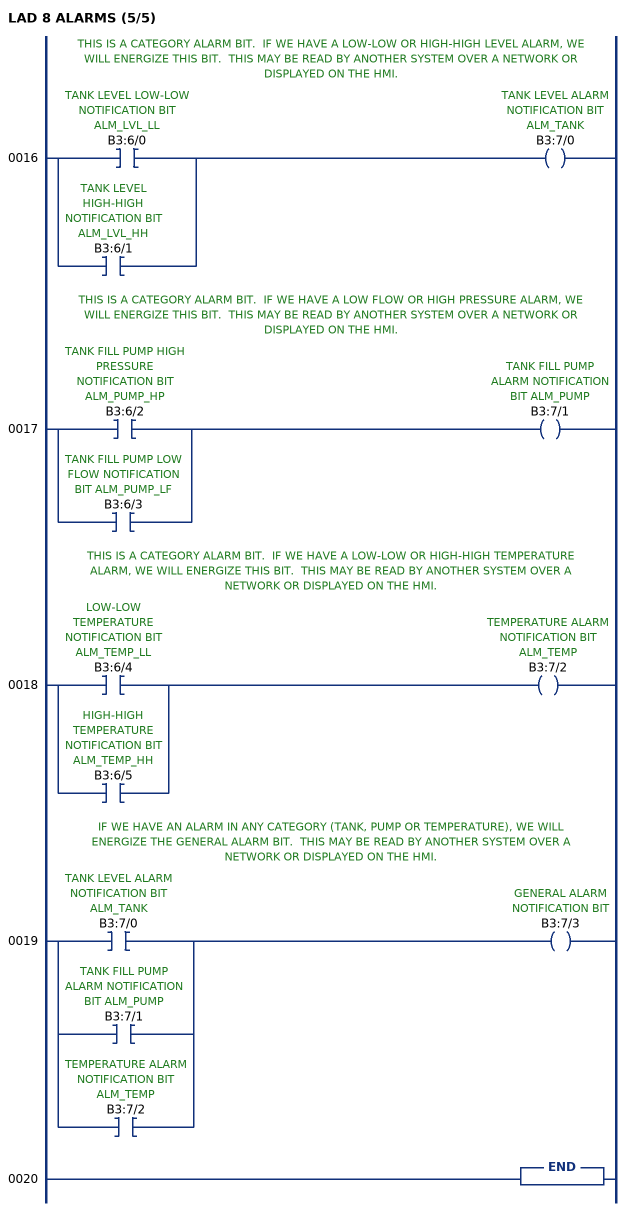
% Rung: 16 %
% THIS IS A CATEGORY ALARM BIT.  IF WE HAVE A LOW-LOW OR HIGH-HIGH LEVEL ALARM, WE WILL ENERGIZE THIS BIT.  THIS MAY BE READ BY ANOTHER SYSTEM OVER A NETWORK OR DISPLAYED ON THE HMI. %
SOR BST XIC B3:6/0 NXB XIC B3:6/1 BND OTE B3:7/0 EOR
%   B3:6/0  ALM_LVL_LL  "TANK LEVEL LOW-LOW NOTIFICATION BIT" %
%   B3:6/1  ALM_LVL_HH  "TANK LEVEL HIGH-HIGH NOTIFICATION BIT" %
%   B3:7/0  ALM_TANK  "TANK LEVEL ALARM NOTIFICATION BIT" %
% Rung: 17 %
% THIS IS A CATEGORY ALARM BIT.  IF WE HAVE A LOW FLOW OR HIGH PRESSURE ALARM, WE WILL ENERGIZE THIS BIT.  THIS MAY BE READ BY ANOTHER SYSTEM OVER A NETWORK OR DISPLAYED ON THE HMI. %
SOR BST XIC B3:6/2 NXB XIC B3:6/3 BND OTE B3:7/1 EOR
%   B3:6/2  ALM_PUMP_HP  "TANK FILL PUMP HIGH PRESSURE NOTIFICATION BIT" %
%   B3:6/3  ALM_PUMP_LF  "TANK FILL PUMP LOW FLOW NOTIFICATION BIT" %
%   B3:7/1  ALM_PUMP  "TANK FILL PUMP ALARM NOTIFICATION BIT" %
% Rung: 18 %
% THIS IS A CATEGORY ALARM BIT.  IF WE HAVE A LOW-LOW OR HIGH-HIGH TEMPERATURE ALARM, WE WILL ENERGIZE THIS BIT.  THIS MAY BE READ BY ANOTHER SYSTEM OVER A NETWORK OR DISPLAYED ON THE HMI. %
SOR BST XIC B3:6/4 NXB XIC B3:6/5 BND OTE B3:7/2 EOR
%   B3:6/4  ALM_TEMP_LL  "LOW-LOW TEMPERATURE NOTIFICATION BIT" %
%   B3:6/5  ALM_TEMP_HH  "HIGH-HIGH TEMPERATURE NOTIFICATION BIT" %
%   B3:7/2  ALM_TEMP  "TEMPERATURE ALARM NOTIFICATION BIT" %
% Rung: 19 %
% IF WE HAVE AN ALARM IN ANY CATEGORY (TANK, PUMP OR TEMPERATURE), WE WILL ENERGIZE THE GENERAL ALARM BIT.  THIS MAY BE READ BY ANOTHER SYSTEM OVER A NETWORK OR DISPLAYED ON THE HMI. %
SOR BST XIC B3:7/0 NXB XIC B3:7/1 NXB XIC B3:7/2 BND OTE B3:7/3 EOR
%   B3:7/0  ALM_TANK  "TANK LEVEL ALARM NOTIFICATION BIT" %
%   B3:7/1  ALM_PUMP  "TANK FILL PUMP ALARM NOTIFICATION BIT" %
%   B3:7/2  ALM_TEMP  "TEMPERATURE ALARM NOTIFICATION BIT" %
%   B3:7/3  "GENERAL ALARM NOTIFICATION BIT" %
% Rung: 20 %
SOR END EOR

LADDER 9 "DISPLAY"
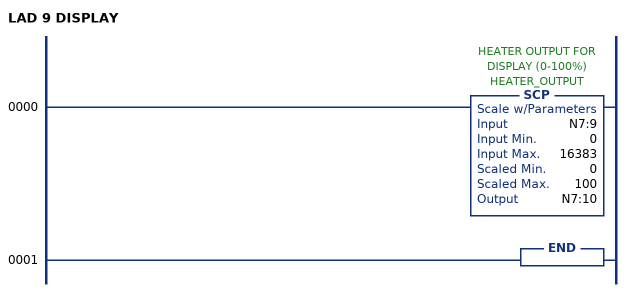
% Rung: 0 %
SOR SCP N7:9 0 16383 0 100 N7:10 EOR
%   N7:9  "HEATER CV" %
%   N7:10  HEATER_OUTPUT  "HEATER OUTPUT FOR DISPLAY (0-100%)" %
% Rung: 1 %
SOR END EOR

COMMENTS NOT ATTACHED TO A CURRENT RUNG
  N7:4: hERE WE LOOK FOR THE PHYSICAL "ON" BUTTON OR THE HMI SYSTEM ON PUSHBUTTON TO BE PRESSED BY THE OPERATOR.  IF AND ONLY IF THE SYSTEM IS IN THE "OFF" MODE, WE CHANGE THE MODE TO ON BY MOVING THE VALUE "1" INTO THE ADDRESS N7:4 (AN ARBITRARILY CHOSEN INTERGER LOCATION TO BE USED THROUGHOUT THE CONTROL LOGIC AND HMI DISPLAYS TO INDICATE SYSTEM MODE).  THE ONS (ONE-SHOT) BLOCK ALLOWS THE OUTPUT TO THE RIGHT TO EXECUTE FOR ONLY ONE SCAN FOR EACH TIME THE CONDITIONS TO THE LEFT OF THE BLOCK ARE ALL TRUE.

DATA TABLE (non-zero values as saved)
DATA B3
% B3:0 % 0X0000 0X001D 0X0500 0X0000 0X0000 0X0008 0X0008 0X000A
DATA T4
% .PRE .ACC %
% T4:0 % 5 0
% T4:1 % 5 0
% T4:2 % 5 0
% T4:3 % 5 0
% T4:4 % 900 0
% T4:5 % 5 0
% T4:6 % 5 5
% T4:7 % 5 0
DATA N7
% N7:0 % 15 20 80 90 2 20 90 120 105 0
% N7:10 % 0 2
DATA F8
% F8:0 % 18.31166 104.6621 0
